(* IEC 61131-3 sources: volt/packages/volt-lsp-iec/test-corpus/bakon-nano/Device/Plc Logic/Application/POUs/FunctionBlocksDRV, 3 files *)

(* ---- DRV_AGM_IO.pou ---- *)
FUNCTION_BLOCK DRV_AGM_IO		(* Depending on ProductType start AGM *)
VAR
	TP_Test: TP;
	TP_Reset: TP;
END_VAR

VAR_INPUT
	I_bCMD_Enable			: BOOL;
	I_bCMD_Start				: BOOL;
	I_bCMD_Test				: BOOL;	(* Manual command *)
	I_bCMD_Reset			: BOOL;	(* Manual command *)
END_VAR

VAR_IN_OUT
	Q_bStart_AGM			: BOOL;
	Q_bTest_AGM				: BOOL;
END_VAR

%LANGUAGE ST
IF NOT I_bCMD_Enable THEN
	Q_bStart_AGM		:=FALSE;
ELSE

	(* Reset errors *)
	TP_Reset(IN:=I_bCMD_REset , PT:=T#200ms);

(**************************************************************************************************************************)
	(* Create test pulse *)
	TP_Test(IN:=I_bCMD_Test , PT:=T#800ms);

(**************************************************************************************************************************)
	(* Execute command  *)
	IF	I_bCMD_Start  OR TP_Reset.Q
	OR TP_Test.Q //Added because of I/O control of AGM
	THEN
		Q_bStart_AGM		:= TRUE;
	ELSE
		Q_bStart_AGM		:= FALSE;
	END_IF

	IF TP_Test.Q THEN
		Q_bTest_AGM := TRUE;
	ELSE
		Q_bTest_AGM := FALSE;
	END_IF
END_IF

END_FUNCTION_BLOCK

(* ---- DRV_CYL1C2D_SafeEnd.pou ---- *)
FUNCTION_BLOCK DRV_CYL1C2D_SafeEnd
VAR_INPUT
	I_bCylEndPos					: BOOL;	(* Sensor cylinder is at end position *)
	I_bCylZeroPos				: BOOL;	(* Sensor cylinder is at zero position *)
	I_bSafeEndOK					: BOOL;	(* Safety sensor from Pilz, used to block the alarm and to block the output *)
	I_sControl						: sCYL_Control;
	I_rTimeOut					: REAL;	(* Time in seconds *)
END_VAR
VAR_IN_OUT
	DRV_ERR_CylEndPos		: BOOL;
	DRV_ERR_CylZeroPos		: BOOL;
	DRV_ERR_CylMultiple		: BOOL;
	DRV_ERR_SafetyNOK		: BOOL;
END_VAR
VAR_OUTPUT
	Q_sStatus						: sCYL_Status;
	Q_bCylToEndPos				: BOOL;
	Q_bCylToZeroPos				: BOOL;
END_VAR
VAR
	DRV_TON1					: TON;
	bCylToEndPos				: BOOL;	(* Memory bit *)
	bCylToZeroPos				: BOOL;	(* Memory bit *)
END_VAR
%LANGUAGE ST
(*************************************************************************
 * HISTORY
 *************************************************************************
 * Update  : 0.00
 * Author  :
 * Changes :
 *************************************************************************)

(* Reset errors *)
IF I_sControl.bErrorReset THEN
	DRV_ERR_CylEndPos		:= FALSE;
	DRV_ERR_CylZeroPos		:= FALSE;
	DRV_ERR_CylMultiple		:= FALSE;
	DRV_ERR_SafetyNOK		:= FALSE;
	DRV_TON1(IN:=FALSE);
END_IF

(* In target bit *)
Q_sStatus.bPosInTarget	:= 		(bCylToEndPos AND I_bCylEndPos AND NOT I_bCylZeroPos)
								OR	(NOT bCylToEndPos AND I_bCylZeroPos AND NOT I_bCylEndPos);

(* Actual position *)
IF I_bCylEndPos THEN
	Q_sStatus.rActualPosition := 1;
ELSIF I_bCylZeroPos THEN
	Q_sStatus.rActualPosition := 0;
ELSE
	Q_sStatus.rActualPosition := -1;
END_IF

IF		NOT I_sControl.bPosExecute
	AND NOT I_sControl.bManual
THEN
	DRV_TON1(IN:=FALSE);
	Q_sStatus.bPosDone := FALSE;
	IF	I_bCylEndPos THEN
		bCylToEndPos := TRUE;
	ELSIF	I_bCylZeroPos THEN
		bCylToEndPos := FALSE;
	END_IF
	//DRV_ERR_SafetyNOK := FALSE;
ELSE

	(* Execute command *)
	IF		(I_sControl.bPosExecute AND I_sControl.rTargetPosition = 1)
		OR	(I_sControl.bManual AND I_sControl.bManualPos AND NOT I_sControl.bManualNeg AND I_bSafeEndOK)
	THEN
		bCylToZeroPos	:= FALSE;
		bCylToEndPos		:= I_bSafeEndOK;
		DRV_ERR_SafetyNOK := NOT I_bSafeEndOK;
	END_IF

	IF		(I_sControl.bPosExecute AND I_sControl.rTargetPosition = 0)
		OR	(I_sControl.bManual AND I_sControl.bManualNeg AND NOT I_sControl.bManualPos)
	THEN
		bCylToEndPos		:= FALSE;
		bCylToZeroPos		:= TRUE;
		//DRV_ERR_SafetyNOK := NOT I_bSafeEndOK;
	END_IF

	(* Generate errors *)
	// changed OR	(NOT bCylToEndPos AND NOT I_bCylZeroPos), because of otherwise not working error when sent down
	DRV_TON1(	IN:=		(bCylToEndPos AND NOT I_bCylEndPos AND I_bSafeEndOK)
						OR	(bCylToZeroPos AND NOT I_bCylZeroPos),
				PT:=	REAL_TO_TIME(1000 * I_rTimeOut));	(* time in seconds *)

	(* TimeOut cylinder to end position *)
	IF DRV_TON1.Q AND bCylToEndPos AND NOT I_bCylEndPos THEN
		DRV_ERR_CylEndPos	:= TRUE;
	END_IF

	(* TimeOut cylinder to Zero position *)
	IF DRV_TON1.Q AND bCylToZeroPos AND NOT I_bCylZeroPos THEN
		DRV_ERR_CylZeroPos	:= TRUE;
	END_IF

	Q_sStatus.bPosDone :=	((I_sControl.rTargetPosition = 1) AND I_bCylEndPos AND NOT(I_bCylZeroPos))
							OR	((I_sControl.rTargetPosition = 0) AND I_bCylZeroPos AND NOT(I_bCylEndPos));

END_IF

(* Detection error *)
IF I_bCylEndPos AND I_bCylZeroPos THEN
	DRV_ERR_CylMultiple	:= TRUE;
END_IF

(* Cylinder control *)
Q_bCylToEndPos := bCylToEndPos AND (I_bSafeEndOK OR I_bCylEndPos);
Q_bCylToZeroPos := bCylToZeroPos AND (I_bSafeEndOK OR I_bCylZeroPos);

END_FUNCTION_BLOCK

(* ---- KC_AxisBasics.pou ---- *)
FUNCTION_BLOCK KC_AxisBasics
VAR_INPUT
	AxisControl						:KC_AxisBasicsControl;
	strHomingParameters				:L_MC1P_HomeParameter;
	bEnableSWLimits					:BOOL;
	bEnableHWLimits					:BOOL;
	xIgnorePosLimit					:BOOL;
	I_bVirtual						:BOOL;
	lrHomePosition					:LREAL;
	I_lrTorqueLimitPos_Value		:LREAL;
	I_lrTorqueLimitNeg_Value		:LREAL;
END_VAR

VAR_IN_OUT
	AxisName						:AXIS_REF;
	//AxisEncoder					: AXIS_REF_ETC_DS402_CS_LENZE;

END_VAR

VAR_OUTPUT
	AxisStatus						:KC_AxisBasicsStatus;
END_VAR

VAR
	dInputs : DWORD;
	AxisBasic1: L_MC1P_AxisBasicControl;
	AxisTorquelimit	: L_MC1P_SetTorqueLimit;
	AxisHWLimits : L_MC1P_HWLimitSwitchInterface;
	AxisCInh : L_MC1P_CinhHandling;
	bRegulatorOn : BOOL;
	bPowerHold : BOOL;
	timeReg : TOF;
	timeReg2 : TOF;
END_VAR

%LANGUAGE ST
(* Torque settings *)
AxisTorquelimit(
	Axis:= AxisName,
	xEnable:= AxisName.xCommunicationOK,
	xSetTorqueLimitPos:= TRUE,
	lrTorqueLimitPos:= I_lrTorqueLimitPos_Value,
	xSetTorqueLimitNeg:= TRUE,
	lrTorqueLimitNeg:= I_lrTorqueLimitNeg_Value,
	xTorqueInputAsPercent:= TRUE,
	xBusy=> ,
	xError=> ,
	eErrorID=> );

(*Hardware limits*)
dInputs := L_MC1P_GetDigInputsFromDrive(Axis:= AxisName); //Bit 16 en 17 zijn de Inputs
(*Falling Trigger van Start signaal als stop signaal*)

AxisHWLimits(
	Axis:= AxisName,
	xEnable:= bEnableHWLimits,
	xLimitSwitchPos:= NOT dInputs.16 AND NOT xIgnorePosLimit,
	xLimitSwitchNeg:= NOT dInputs.17,
	xOverwriteOtherSources:= ,
	xBusy=> ,
	xError=> ,
	eErrorID=> );

//Emergency stop handling
AxisCInh(
	Axis:= AxisName,
	xEnable:= TRUE,
	xStayInLastState:= TRUE,
);

AxisBasic1(
	Axis:= AxisName,
	xEnableInternalControl:= TRUE,
	xRegulatorOn:= (AxisControl.bEnableDrive AND g_bDI_ES_DirectOK) OR timereg.Q,// OR (bRegulatorOn), ,
	xResetError:= AxisControl.bResetError,// OR (AxisBasic1.xResetError AND NOT AxisBasic1.xFunDone), ,
	xEnablePositive:= TRUE,
	xEnableNegative:= TRUE,
	xDisableSWLimit:= ,
	lrOverride:= ,
	lrOverrideAcc:= ,
	lrOverrideJerk:= ,
	xStop:= NOT g_bDI_ES_DirectOK AND timeReg.Q AND NOT I_bVirtual,(*Todo True = Ga in Quickstop*)
	lrStopDec:= AxisControl.lrQuickStopDec,	// 20000,
	lrStopJerk:= ,
	xJoggingPos:= AxisControl.bManualJogPos,
	xJoggingNeg:= AxisControl.bManualJogNeg,
	lrJoggingSetVel:= AxisControl.lrVelocity,
	lrJoggingSetAcc:= AxisControl.lrAcceleration,
	lrJoggingSetDec:= AxisControl.lrDeceleration,
	lrJoggingSetJerk:= ,
	xContinuousUpdate:= ,
	xMoveVelExecute:= ,
	xMoveAbsExecute:= AxisControl.bPosABSPosition,
	xMoveRelExecute:= AxisControl.bPosRelPosition,
	xHalt:= ,
	lrSetPos_Dist:= AxisControl.lrPosition,
	lrSetVel:= AxisControl.lrVelocity,
	lrSetAcc:= AxisControl.lrAcceleration,
	lrSetDec:= AxisControl.lrDeceleration,
	lrSetJerk:= ,
	eSetDirection:= ,
	xHomeExecute:= AxisControl.bStartHoming,
	lrHomePosition:= lrHomePosition,
	xUseHomeExtParameter:= TRUE,
	scHomeExtParameter:= strHomingParameters,
	scHomeExtTP:= ,
	xHomeAbsSwitch:= ,
	xInternalControlActive=> ,
	xError=> AxisStatus.xError,
	eErrorID=> AxisStatus.eErrorID,
	xFunBusy=> ,
	xFunDone=> ,
	xFunCommandAborted=> ,
	eFunStateAct=> ,
	eControlMode=> ,
	xIsHomed=> AxisStatus.bHomePositionAvailable,
	xHwLimitSwitchNeg=> AxisStatus.bLimitNeg,
	xHwLimitSwitchPos=> AxisStatus.bLimitPos,
	xSwLimitEnabled=> ,
	xSwLimitSwitchNeg=> ,
	xSwLimitSwitchPos=> ,
	eAxisType=> ,
	eAxisState=> AxisStatus.eStateAxis,
	xAxisReady=> AxisStatus.bDriveReady,
	xAxisEnabled=> ,
	xAxisWarning=> ,
	xAxisError=> AxisStatus.xAxisError,
	eAxisErrorID=> AxisStatus.eAxisErrorID,
	xDriveWarning=> AxisStatus.bDriveWarning,
	xDriveError=> AxisStatus.xDriveError,
	dwDriveErrorID=> AxisStatus.dwDriveErrorID,
	lrActPos=> AxisStatus.lrActPosition,
	lrActVel=> AxisStatus.lrActVelocity,
	lrSetPosOut=> ,
	lrSetVelOut=> ,
	lrActFollowingError=> AxisStatus.lrActFollowError,
	xConstantVelocity=> ,
	xAccelerating=> ,
	xDecelerating=> ,
	xDirectionPositive=> ,
	xDirectionNegative=> ,
	xInPosition=> ,
	xAxisAvailable=> ,
	xStandstillSetVelocity=> ,
	xStandstillActVelocity=> ,
	xAxisReadyToSwitchOn=> ,
	xAxisReadyForMotion=> );

	AxisStatus.bDriveEnabled := AxisBasic1.xAxisEnabled AND AxisBasic1.xAxisReadyForMotion;
	AxisStatus.bHomingDone := AxisControl.bStartHoming AND AxisBasic1.xFunDone;
	AxisStatus.bHomingBusy := AxisControl.bStartHoming AND AxisBasic1.xFunBusy;
	AxisStatus.bManualBusy := (AxisControl.bManualJogPos OR AxisControl.bManualJogNeg) AND AxisBasic1.xFunBusy;
	AxisStatus.bMoveAbsDone := AxisControl.bPosAbsPosition AND AxisBasic1.xFunDone;
	AxisStatus.bMoveRelDone := AxisControl.bPosRelPosition AND AxisBasic1.xFunDone;
	AxisStatus.bDigIn1 :=  dInputs.16;
	AxisStatus.bDigIn2 :=  dInputs.17;

	bRegulatorOn := AxisBasic1.xRegulatorOn AND (AxisBasic1.eAxisState > L_MC1P_AXIS_STATE.StandStill);
	bPowerHold := AxisBasic1.xRegulatorOn AND AxisBasic1.eAxisState > L_MC1P_AXIS_STATE.Stopping;
	timeReg(IN:= AxisControl.bEnableDrive AND g_bDI_ES_DirectOK, PT:=T#100MS);
	timeReg2(IN:= AxisControl.bEnableDrive AND g_bDI_ES_DirectOK, PT:=T#160MS);

END_FUNCTION_BLOCK
